// TIA Portal V18 export
DATA_BLOCK "PalletRelease"   // DB9001
{ S7_Optimized_Access := 'FALSE' }
VERSION : 0.1
// stored: AutoNumber false, DBAccessibleFromOPCUA true, DBAccessibleFromWebserver true, IsOnlyStoredInLoadMemory false, IsWriteProtectedInAS false
   VAR
      Buffer : Struct
         AskPallet : Bool;
         UnloadFlag : Bool;
      END_STRUCT;
      LaserMarking : Struct
         AskPallet : Bool;
         UnloadFlag : Bool;
      END_STRUCT;
      Print : Struct
         AskPallet : Bool;
         UnloadFlag : Bool;
      END_STRUCT;
      Spare : Struct
         AskPallet : Bool;
         UnloadFlag : Bool;
      END_STRUCT;
      Spare2 : Struct
         AskPallet : Bool;
         UnloadFlag : Bool;
      END_STRUCT;
      "Time" : Array[0..1] of TOF_TIME;
      LaserMarkingBuffer : "LaserMarkingBuffer";
   END_VAR
BEGIN
END_DATA_BLOCK
